Staubli VAL3: chinese.pjx

Parameters version=s7.6 stackSize=5000 millimeterUnit=true
Program file=BuildTitle.pgx
Program file=Menu.pgx
Program file=Page.pgx
Program file=start.pgx
Program file=stop.pgx
Data file=chinese.dtx
Library alias=up path=Disk://Tracking/Tools/userPage/userPage.pjx
